// TwinCAT 3 PLC project Heatpump
// ProgramVersion: 3.1.4026.11
// libraries:
//   Tc2_Math, * (Beckhoff Automation GmbH)
//   Tc2_Standard, * (Beckhoff Automation GmbH)
//   Tc2_System, * (Beckhoff Automation GmbH)
//   Tc2_Utilities, * (Beckhoff Automation GmbH)
// project tree:
//   DUTs/ E_Event.TcDUT, E_EventType.TcDUT, E_LogType.TcDUT, E_Severity.TcDUT, E_State.TcDUT, ST_ConfigValues.TcDUT, ST_Event.TcDUT, ST_Events.TcDUT, ST_ErrorEvents.TcDUT, ST_LogBuffer.TcDUT, ST_LogEntry.TcDUT, ST_WarningEvents.TcDUT, ST_SensorRaw.TcDUT, ST_Actor.TcDUT, ST_FailureMessage.TcDUT, ST_Incident.TcDUT, ST_ProcessData.TcDUT, E_FailureLevel.TcDUT, ST_Sensor.TcDUT
//   GVLs/ GVL.TcGVL
//   / PlcTask.TcTTO
//   POUs/ FB_CoolDownState.TcPOU, FB_ErrorState.TcPOU, FB_IdleState.TcPOU, FB_OffState.TcPOU, FB_ProcessData.TcPOU, FB_RunningState.TcPOU, FB_StartWaterFlowState.TcPOU, FB_StateMachine.TcPOU, I_State.TcIO, MAIN.TcPOU
//   POUs/utils/ calculateTargetTemperatureOn.TcPOU, calculateTargetTemperatureOff.TcPOU, convertTimerToDisplayValue.TcPOU, isVentilOpen.TcPOU, LogMessage.TcPOU, setEventInfo.TcPOU, resetApplication.TcPOU, ScaleAndRound.TcPOU, ScaleAndRoundString.TcPOU, switchWaterVentil.TcPOU, toErrorText.TcPOU, toggleIntermediateCircuitPump.TcPOU, togglePvBoost.TcPOU, transitionToErrorState.TcPOU, clearErrorList.TcPOU, updateEventWithTimestamp.TcPOU, UpdateLogTimestampWithSystemTime.TcPOU
// real-time tasks:
//   TASK PlcTask: cycle T#10ms, priority 1, ADS port 350
// I/O:
//   DEVICE Gerät 1 (EtherCAT), AmsNetId 5.124.202.224.2.1
//     Klemme 10 (EK1200) [EK1200-5000 EtherCAT Netzteil (2A E-Bus)]
//       Klemme 2 (EL3152) [EL3152 2K. Ana. Eingang 4-20mA]
//       Klemme 3 (EL2004) [EL2004 4K. Dig. Ausgang 24V, 0.5A]
//       Klemme 4 (EL3204) [EL3204 4K. Ana. Eingang PT100 (RTD)]
//       Klemme 5 (EL3102) [EL3102 2K. Ana. Eingang +/-10V, Diff.]
//       Klemme 6 (EL1008) [EL1008 8K. Dig. Eingang 24V, 3ms]
//       Klemme 18 (EL1008) [EL1008 8K. Dig. Eingang 24V, 3ms]
//       Klemme 7 (EL3204) [EL3204 4K. Ana. Eingang PT100 (RTD)]
//       Klemme 9 (EL2622) [EL2622 2K. Relais Ausgang, Schließer (230V AC / 30V DC)]
//       Klemme 8 (EL2622) [EL2622 2K. Relais Ausgang, Schließer (230V AC / 30V DC)]
//       Klemme 19 (EL3204) [EL3204 4K. Ana. Eingang PT100 (RTD)]
//       Klemme 20 (EL9011) [EL9011 Endklemme]
// variable links:
//   Heatpump/Heatpump Instance <-> Device 1 (EtherCAT)/Term 10 (EK1200)/Term 18 (EL1008)
//     PlcTask Inputs/MAIN.pd.incident.incidentFlowIntermediateCircuit <-> Channel 1/Input
//   Heatpump/Heatpump Instance <-> Device 1 (EtherCAT)/Term 10 (EK1200)/Term 19 (EL3204)
//     PlcTask Inputs/MAIN.fbProcessdata.sensorRaw.temperatureSourceWaterIn <-> RTD Inputs Channel 1/Value
//     PlcTask Inputs/MAIN.fbProcessdata.sensorRaw.temperatureSourceWaterOut <-> RTD Inputs Channel 2/Value
//   Heatpump/Heatpump Instance <-> Device 1 (EtherCAT)/Term 10 (EK1200)/Term 2 (EL3152)
//     PlcTask Inputs/MAIN.fbProcessdata.sensorRaw.pressureHigh <-> Channel 1/Value
//     PlcTask Inputs/MAIN.fbProcessdata.sensorRaw.pressureLow <-> Channel 2/Value
//   Heatpump/Heatpump Instance <-> Device 1 (EtherCAT)/Term 10 (EK1200)/Term 3 (EL2004)
//     PlcTask Outputs/MAIN.pd.actor.operatingStateCompressor <-> Channel 1/Output
//     PlcTask Outputs/MAIN.pd.actor.operatingStateLed <-> Channel 3/Output
//     PlcTask Outputs/MAIN.pd.actor.operatingStateWaterPump <-> Channel 2/Output
//   Heatpump/Heatpump Instance <-> Device 1 (EtherCAT)/Term 10 (EK1200)/Term 4 (EL3204)
//     PlcTask Inputs/MAIN.fbProcessdata.sensorRaw.temperatureEvaporatingIn <-> RTD Inputs Channel 2/Value
//     PlcTask Inputs/MAIN.fbProcessdata.sensorRaw.temperatureEvaporatingOut <-> RTD Inputs Channel 1/Value
//     PlcTask Inputs/MAIN.fbProcessdata.sensorRaw.temperatureFlow <-> RTD Inputs Channel 3/Value
//     PlcTask Inputs/MAIN.fbProcessdata.sensorRaw.temperatureReturn <-> RTD Inputs Channel 4/Value
//   Heatpump/Heatpump Instance <-> Device 1 (EtherCAT)/Term 10 (EK1200)/Term 5 (EL3102)
//     PlcTask Inputs/MAIN.fbProcessdata.sensorRaw.pressureDifferenceEvaporator <-> Channel 1/Value
//   Heatpump/Heatpump Instance <-> Device 1 (EtherCAT)/Term 10 (EK1200)/Term 6 (EL1008)
//     PlcTask Inputs/MAIN.pd.incident.alarmExpansionValve <-> Channel 3/Input
//     PlcTask Inputs/MAIN.pd.incident.incidentCompressor <-> Channel 5/Input
//     PlcTask Inputs/MAIN.pd.incident.incidentHighPressure <-> Channel 7/Input
//     PlcTask Inputs/MAIN.pd.incident.incidentLowPressure <-> Channel 8/Input
//     PlcTask Inputs/MAIN.pd.incident.incidentWaterFlow <-> Channel 6/Input
//     PlcTask Inputs/MAIN.pd.sensor.boilerHeatRequest <-> Channel 2/Input
//     PlcTask Inputs/MAIN.pd.sensor.photovoltaicSurplus <-> Channel 4/Input
//     PlcTask Inputs/MAIN.pd.sensor.userConfirmation <-> Channel 1/Input
//   Heatpump/Heatpump Instance <-> Device 1 (EtherCAT)/Term 10 (EK1200)/Term 7 (EL3204)
//     PlcTask Inputs/MAIN.fbProcessdata.sensorRaw.boilerTemperature <-> RTD Inputs Channel 4/Value
//     PlcTask Inputs/MAIN.fbProcessdata.sensorRaw.bufferMiddleTemperature <-> RTD Inputs Channel 2/Value
//     PlcTask Inputs/MAIN.fbProcessdata.sensorRaw.bufferTopTemperature <-> RTD Inputs Channel 3/Value
//     PlcTask Inputs/MAIN.fbProcessdata.sensorRaw.temperatureOverheatedGas <-> RTD Inputs Channel 1/Value
//   Heatpump/Heatpump Instance <-> Device 1 (EtherCAT)/Term 10 (EK1200)/Term 8 (EL2622)
//     PlcTask Outputs/MAIN.pd.actor.operatingStateIntermediateCircuitPump <-> Channel 1/Output
//   Heatpump/Heatpump Instance <-> Device 1 (EtherCAT)/Term 10 (EK1200)/Term 9 (EL2622)
//     PlcTask Outputs/MAIN.pd.actor.closeFlowVentil <-> Channel 1/Output
//     PlcTask Outputs/MAIN.pd.actor.openFlowVentil <-> Channel 2/Output

CONFIGURATION Heatpump
    RESOURCE PLC ON TwinCAT3
        TASK PlcTask(INTERVAL := T#1ms, PRIORITY := 4);
        PROGRAM MAIN WITH PlcTask : MAIN;
    END_RESOURCE
END_CONFIGURATION

// ---- DUTs/E_Event.TcDUT
{attribute 'qualified_only'}
{attribute 'strict'}
TYPE E_Event :
(
	SwitchOn := 0,
	SwitchOff := 1,
	HeatIsRequested := 2,
	HeatTemperaturreached := 3,
	CooledDown := 4,
	Confirmed := 5
);
END_TYPE

// ---- DUTs/E_EventType.TcDUT
{attribute 'qualified_only'}
{attribute 'strict'}
TYPE E_EventType :
(
	None								:= 0,
	(* Normal StateMachine changes *)	
	SwitchOn 							:= 1,
	SwitchOff 							:= 2,
	HeatIsRequested 					:= 3,
	TargetTemperatureReached 			:= 4,
	CooledDown 							:= 5,
	Confirm 							:= 6,
	minWaterFlowReached					:= 7,
	
	(* Errors *)
	PressureDiffEvaporatorTooHigh		:= 101,
	EvaporatingTemperatureTooLow		:= 102,
	EvaporatingFlowRateTooLow			:= 103,
	LowPressureRefrigerationThermostat	:= 104,
	HighPressureRefrigerationThermostat	:= 105,
	MotorProtectionTriggered			:= 106,
	ExpansionValveTriggered				:= 107,
	IntermediateCircuitFlowRateTooLow	:= 108,
	LowPressureRefrigerationCalc		:= 109,
	TemperatureSourceWaterOutMinTooLow  := 110,
		
	(* Warnings *)
	HighPressureRefrigerationCalc		:= 202,
	WaterTankLevelTooLow				:= 203,
	WaterTankDataMissing				:= 204
);
END_TYPE

// ---- DUTs/E_LogType.TcDUT
{attribute 'qualified_only'}
{attribute 'strict'}
TYPE E_LogType :
(
    INFO := 0,
    WARNING := 1,
    ERROR := 2
);
END_TYPE

// ---- DUTs/E_Severity.TcDUT
{attribute 'qualified_only'}
{attribute 'strict'}
TYPE E_Severity :
(
	Error := 0,
	Warning := 1,
	Event := 2
);
END_TYPE

// ---- DUTs/E_State.TcDUT
{attribute 'qualified_only'}
{attribute 'strict'}
TYPE E_State :
(
	OFF := 0,
	IDLE := 1,
	START_WATER_FLOW := 2,
	RUNNING := 3,
	COOLDOWN := 4,
    ERROR := 5
);
END_TYPE

// ---- DUTs/ST_ConfigValues.TcDUT
TYPE ST_ConfigValues :
STRUCT	
	targetTemperatureOn 			:	REAL	:= 	33; 	// Einschalttemperatur bei deren Unterschreiten die Waermepumpe eingeschaltet wird
	targetTemperatureOnPV 			:	REAL	:= 	40; 	// Bei PV-Überschuss: Einschalttemperatur bei deren Unterschreiten die Waermepumpe eingeschaltet wird
	targetTemperatureOff 			:	REAL	:= 	41; 	// Auschaltemperatur bei deren Ueberschreiten die Waermepume ausgeschaltet wird	
	targetTemperatureOffPV			:	REAL	:= 	50; 	// Bei PV-Überschuss: Auschaltemperatur bei deren Ueberschreiten die Waermepume ausgeschaltet wird	
	maxReturnTemperature			:	REAL	:= 	53; 	// Schaltet aus / nicht ein, falls Rücklauf Temperatur zu hoch, z.B. wenn Holzkessel heizt
	minIdleSec 						:	TIME 	:= 	T#10M;	// Minimale Auschalt-Dauer (verhindert haeufiges Einschalten) [Minuten]
	temperatureDiffBacklashOff 		:	REAL	:= 	1.0; 	// Temperaturdifferenz zwischen Vorlauf und Rücklauf, bei dessen Unterschreiten die Wasserpumpe ausgeschaltet wird
	temperatureDiffBoilerLaden 		:	REAL	:= 	4.0; 	// Temperaturdifferenz zwischen Puffer oben und Boiler, die unterschritten sein muss, damit die Wärmepumpe einschaltet.

	// Limits*)
	pressureHighMax 				:	REAL	:= 	16; 	// Maximaler Druck auf der Hochdruckseite [bar]
	pressureLowMin 					:	REAL	:= 	0.4; 	// Minimaler Druck auf der Niederdruckseite [bar]. Entspricht -5°C. Falls niedriger deutet dies auf ein Kältemittel-Leck hin 
	pressureDifferenceEvaporatorMax :	REAL 	:= 	45;		// Maximaler Druckverlust des Verdampfer-Wärmetauschers [mbar]
	evaporatingTemperatureOutMin 	:	REAL 	:=	1.0; 	// Minimale Temperatur am Austritt des Verdampfer-Wärmetausschers. Triplepunkt des Wassers. [°C]	
	temperatureSourceWaterOutMin	:	REAL 	:=	2.3;  	// Minimale Temperatur am Quellasser-Austritt des Zwischenkreis-Wärmetausschers. Triplepunkt des Wassers. [°C]
END_STRUCT
END_TYPE

// ---- DUTs/ST_Event.TcDUT
TYPE ST_Event :
STRUCT
	eventType		: E_EventType := E_EventType.None;
	severity 		: E_Severity := E_Severity.Event;
	isTriggered		: BOOL := FALSE;
	isSelfHealing   : BOOL := FALSE;  	// selbst heilend: Nach einem Error und automatischem Beheben der Ursache startet die WP wieder
	message	 		: STRING(255);
	timestamp 		: DATE_AND_TIME;
END_STRUCT
END_TYPE

// ---- DUTs/ST_Events.TcDUT
TYPE ST_Events :
STRUCT
	(* Normal StateMachine changes *)
	switchOff 							: ST_Event := (eventType := E_EventType.SwitchOff);  
	switchOn 							: ST_Event := (eventType := E_EventType.SwitchOn);  
	confirmed							: ST_Event := (eventType := E_EventType.Confirm);
	heatIsRequested 					: ST_Event := (eventType := E_EventType.HeatIsRequested);  
	targetTemperatureReached			: ST_Event := (eventType := E_EventType.TargetTemperatureReached);
	cooledDown							: ST_Event := (eventType := E_EventType.CooledDown);
	minWaterFlowReached					: ST_Event := (eventType := E_EventType.MinWaterFlowReached);
		
	(* Errors *)
     errorEvents						: ST_ErrorEvents; 
	 errorsDetected						: BOOL := FALSE;

	(* Warnings *)
	warningEvents						:ST_WarningEvents;
END_STRUCT
END_TYPE

// ---- DUTs/ST_ErrorEvents.TcDUT
TYPE ST_ErrorEvents :
	STRUCT
		(* Errors *)
		PressureDiffEvaporatorTooHigh		: ST_Event := (eventType := E_EventType.PressureDiffEvaporatorTooHigh, isSelfHealing:=FALSE, severity:= E_Severity.Error, message := 'Druckdifferenz am Verdampfer zu hoch. Einfriergefahr');  
		EvaporatingTemperatureTooLow		: ST_Event := (eventType := E_EventType.EvaporatingTemperatureTooLow, isSelfHealing:=TRUE, severity:= E_Severity.Error, message := 'Autrittstemperatur zu niedrig');  
		EvaporatingFlowRateTooLow			: ST_Event := (eventType := E_EventType.EvaporatingFlowRateTooLow, isSelfHealing:=TRUE, severity:= E_Severity.Error, message := 'Durchflussmenge zu niedrig');  
		LowPressureRefrigerationThermostat	: ST_Event := (eventType := E_EventType.LowPressureRefrigerationThermostat, isSelfHealing:=FALSE, severity:= E_Severity.Error, message := 'Thermostat: Niederdruck zu niedrig');  
		HighPressureRefrigerationThermostat	: ST_Event := (eventType := E_EventType.HighPressureRefrigerationThermostat, isSelfHealing:=FALSE, severity:= E_Severity.Error, message := 'Thermostat: Hochdruck zu hoch');  
		MotorProtectionTriggered			: ST_Event := (eventType := E_EventType.MotorProtectionTriggered, isSelfHealing:=FALSE, severity:= E_Severity.Error, message := 'Motorschutzschalter hat ausgelöst');  
		ExpansionValveTriggered				: ST_Event := (eventType := E_EventType.ExpansionValveTriggered, isSelfHealing:=FALSE, severity:= E_Severity.Error, message := 'Expansionsventil ausgelöst');
		IntermediateCircuitFlowRateTooLow	: ST_Event := (eventType := E_EventType.IntermediateCircuitFlowRateTooLow, isSelfHealing:=TRUE, severity:= E_Severity.Error, message := 'Sole Durchflussmenge im Zwischenkreis zu niedrig');
		LowPressureRefrigerationCalc		: ST_Event := (eventType := E_EventType.LowPressureRefrigerationCalc, isSelfHealing:=FALSE, severity:= E_Severity.Error, message := 'Sensor: Niederdruck zu niedrig');  
		TemperatureSourceWaterOutMinTooLow	: ST_Event := (eventType := E_EventType.TemperatureSourceWaterOutMinTooLow, isSelfHealing:=TRUE, severity:= E_Severity.Error, message := 'Quellwasser-Autrittstemperatur zu niedrig. Einfriergefahr');  
	END_STRUCT
END_TYPE

// ---- DUTs/ST_LogBuffer.TcDUT
TYPE ST_LogBuffer :
STRUCT
    aEntries : ARRAY[1..100] OF ST_LogEntry;
END_STRUCT
END_TYPE

// ---- DUTs/ST_LogEntry.TcDUT
TYPE ST_LogEntry :
STRUCT
    sMessage : STRING(255);
    dtTimestamp : DATE_AND_TIME;
    eType : E_LogType;
	sTypeName : STRING(20);
END_STRUCT
END_TYPE

// ---- DUTs/ST_WarningEvents.TcDUT
TYPE ST_WarningEvents :
STRUCT
	(* Warnings *)
	HighPressureRefrigerationCalc		: ST_Event := (eventType := E_EventType.HighPressureRefrigerationCalc, severity:= E_Severity.Warning, message := 'Sensor: Niederdruck zu hoch');  
	WaterTankLevelTooLow				: ST_Event := (eventType := E_EventType.WaterTankLevelTooLow, severity:= E_Severity.Warning, message := 'Wasserstand des Tanks (Quelle) zu niedrig');  
	WaterTankDataMissing				: ST_Event := (eventType := E_EventType.WaterTankDataMissing, severity:= E_Severity.Warning, message := 'Tanksensor (Quelle) sendet keine Daten mehr');  
END_STRUCT
END_TYPE

// ---- DUTs/ST_SensorRaw.TcDUT
TYPE ST_SensorRaw :
    STRUCT
		(* EL3204 - 1*)
        temperatureEvaporatingOut		AT %I*	: INT;  (* Verdampfungstemperatur in °C (Ausgang) *)
        temperatureEvaporatingIn		AT %I*	: INT;  (* Verdampfungstemperatur in °C (Eingang) *)
        temperatureFlow	 				AT %I*	: INT;  (* Vorlauftemperatur in °C *)
        temperatureReturn				AT %I*	: INT;  (* Rücklauftemperatur in °C *)
		
		(* EL3204 - 2*)
        temperatureOverheatedGas		AT %I*	: INT;  (* Saugtemperatur des überhitzten Gases *)
        bufferTopTemperature			AT %I*	: INT;  (* Temperatur des Puffers oben in °C *)
		bufferMiddleTemperature			AT %I*	: INT;  (* Temperatur des Puffers in der Mitte °C *)	
		boilerTemperature				AT %I*	: INT;  (* Boiler-Temperatur oben °C *)	
		
		(* EL3204 - 3*)
		temperatureSourceWaterIn		AT %I*	: INT;  (* Quellwassertemperatur Eingang in °C *)
		temperatureSourceWaterOut		AT %I*	: INT;  (* Quellwassertemperatur Ausgang in °C *)		

		(* EL3122 - 4-20mA*)
        pressureHigh					AT %I*	: INT;  (* Hochdruck Kältekreis in bar *)
        pressureLow						AT %I*	: INT;  (* Niederdruck Kältekreis in bar *)
		
		(* EL3064 - 0-10V* or EL3102 -  +/-10V *)
        pressureDifferenceEvaporator	AT %I*	: INT;  (* Druckdifferenz im Verdampfer in mbar *)
    END_STRUCT
END_TYPE

// ---- DUTs/ST_Actor.TcDUT
TYPE ST_Actor :
    STRUCT
		(* EL2004 - Digital Out*)
        operatingStateCompressor 				AT %Q* : BOOL := FALSE;  // Status des Verdichters: Ein/Aus
        operatingStateWaterPump 				AT %Q* : BOOL := FALSE;  // Status der Heizungspumpe: Ein/Aus
        operatingStateIntermediateCircuitPump 	AT %Q* : BOOL := FALSE;  // Status der Heizungspumpe: Ein/Aus
		operatingStateLed						AT %Q* : BOOL := FALSE;  // LED am Schaltschrank, die anzeigt ob die Wärmepumpe eingschaltet/bereit ist
		openFlowVentil   						AT %Q* : BOOL := FALSE;  // Wasserventil öffnen
		closeFlowVentil   						AT %Q* : BOOL := FALSE;  // Wasserventil schliessen 
    END_STRUCT
END_TYPE

// ---- DUTs/ST_FailureMessage.TcDUT
TYPE ST_FailureMessage :
    STRUCT
        message: STRING[100];  (* Fehlermeldung *)
        level: E_FailureLevel;  (* Fehlerstufe *)
    END_STRUCT
END_TYPE

// ---- DUTs/ST_Incident.TcDUT
TYPE ST_Incident :
    STRUCT
		// Connected to IO Klemmen		
        alarmExpansionValve				AT %I*			: BOOL;		// Alarm: Elektronisches Expansionsventil - EL1008.3
        incidentCompressor				AT %I*			: BOOL; 	// Störung: Verdichter / Motorschutzschalter - EL1008.5
        incidentWaterFlow				AT %I*			: BOOL; 	// Störung: Quellwasser-Durchfluss zu niedrig - EL1008.6  Achtung!!! invertiert: True bedeutet genug Fluss vorhanden
        incidentFlowIntermediateCircuit	AT %I*			: BOOL; 	// Störung: Durchfluss im Verdampfer (Zwischenkreis) zu niedrig. Achtung!!! invertiert: True bedeutet genug Fluss vorhanden 
        incidentHighPressure			AT %I*			: BOOL; 	// Störung: Hochdruck zu hoch - EL1008.7
        incidentLowPressure				AT %I*			: BOOL; 	// Störung: Niederdruck zu niedrig - EL1008.8 

		// Calculated from Business Logic
        incidentTankLevelTooLow					: BOOL;  // Störung: Wasserstand des Tanks zu niedrig 
        incidentTankSensorDataMissing			: BOOL;  // Störung: Tanksensor sendet keine Daten mehr 
    END_STRUCT
END_TYPE

// ---- DUTs/ST_ProcessData.TcDUT
TYPE ST_ProcessData :
    STRUCT
        id					: STRING[50];  (* Äquivalent zu String in Java *)
        timestamp			: TIME;  (* Äquivalent zu Instant in Java *)
        sensor				: ST_Sensor;  (* Instanz von Sensor *)
        actor				: ST_Actor;  (* Instanz von Actor *)
        incident			: ST_Incident;  (* Instanz von Incident *)
        waitCounter			: INT;  (* Integer *)
        messages			: ARRAY[1..10] OF ST_FailureMessage;  (* Set als Array, maximale Anzahl definieren *)
    END_STRUCT
END_TYPE

// ---- DUTs/E_FailureLevel.TcDUT
{attribute 'qualified_only'}
{attribute 'strict'}
{attribute 'to_string'}
TYPE E_FailureLevel :
( 
    ERROR := 0,
    WARNING := 1,
    INFO := 2
);
END_TYPE

// ---- DUTs/ST_Sensor.TcDUT
TYPE ST_Sensor :
    STRUCT
        temperatureEvaporatingIn				: REAL;  // Verdampfungstemperatur in °C (Eingang)
        temperatureEvaporatingOut				: REAL;  // Verdampfungstemperatur in °C (Ausgang)
        temperatureFlow	 						: REAL;  // Vorlauftemperatur in °C
        temperatureReturn						: REAL;  // Rücklauftemperatur in °C
        bufferTopTemperature					: REAL;  // Temperatur des Puffers oben in °C
        bufferMiddleTemperature					: REAL;  // Temperatur des Puffers in der Mitte °C		
		boilerTemperature						: REAL;  // Boiler-Temperatur oben °C
        temperatureOverheatedGas				: REAL;  // Saugtemperatur des überhitzten Gases
        temperatureSourceWaterIn				: REAL;  // Quellwassertemperatur Eingang in °C
        temperatureSourceWaterOut				: REAL;  // Quellwassertemperatur Ausgang in °C
        pressureHigh							: REAL;  // Hochdruck Kältekreis in bar
        pressureLow								: REAL;  // Niederdruck Kältekreis in bar
        pressureDifferenceEvaporator			: REAL;  // Druckdifferenz im Verdampfer in mbar
        calculatedOverheatTemperature			: REAL;  // Berechnete Überhitzungstemperatur
        boilerHeatRequest				AT %I*	: BOOL;  // Boiler LadePumpe ist eingeschaltet - EL1008.1*)
        userConfirmation				AT %I*	: BOOL;  // Taster für Ein-/Aus-Quittierung - EL1008.2*) 
		photovoltaicSurplus				AT %I*	: BOOL;  // Photovoltaik Überschuss - gemeldet vom PV-WechselrichterEL1008.4*)
		photovoltaicBoost				  		: BOOL;  // Photovoltaik Boost - ist kein Sensor - sondern per Click einschaltbar*)
    END_STRUCT
END_TYPE

// ---- GVLs/GVL.TcGVL
{attribute 'qualified_only'}
VAR_GLOBAL PERSISTENT
	configValues			:   ST_ConfigValues;			// Konfigurationsparaeter - Müssen vom User geändert werden können
END_VAR
VAR_GLOBAL 
	lastErrorsOccurred		:   ARRAY[0..6] OF ST_Event;  	// List of last errors occurred
	g_LogData : ST_LogBuffer;
END_VAR

// ---- POUs/I_State.TcIO
INTERFACE I_State

PROPERTY Description : STRING
GET
END_GET
END_PROPERTY

METHOD ErrorDetected : BOOL
VAR_IN_OUT
	errorEvents		: ST_ErrorEvents;
END_VAR
END_METHOD

METHOD HeatIsRequested : BOOL
VAR_INPUT
END_VAR
END_METHOD

METHOD MinWaterFlowReached : BOOL
VAR_INPUT
END_VAR
END_METHOD

PROPERTY Name : String
GET
END_GET
END_PROPERTY

PROPERTY State : E_State
GET
END_GET
END_PROPERTY

METHOD TargetTemperatureReached : BOOL
VAR_INPUT
END_VAR
END_METHOD

METHOD UserPressedConfirmationButton : BOOL
VAR_INPUT
END_VAR
END_METHOD

METHOD UserPressedSwitchOffButton : BOOL
VAR_INPUT
END_VAR
END_METHOD

METHOD UserPressedSwitchOnButton : BOOL
VAR_INPUT
END_VAR
END_METHOD

METHOD WaterHasCooledDown : BOOL
VAR_INPUT
END_VAR
END_METHOD

END_INTERFACE

// ---- POUs/MAIN.TcPOU
PROGRAM MAIN
VAR
	fbStateMachine				:	FB_StateMachine;
	fbProcessdata				:   FB_Processdata;
	pd 							: 	ST_ProcessData;	
END_VAR

fbProcessdata(pd := pd);

fbStateMachine(pd := pd);

END_PROGRAM

// ---- POUs/FB_StateMachine.TcPOU
FUNCTION_BLOCK FB_StateMachine
VAR_INPUT	
	pd 							: 	REFERENCE TO ST_ProcessData;
END_VAR
VAR_OUTPUT
	iState						:	I_State := fbOffState;	
	events						:	ST_Events();
	defaultEvents 				: 	ST_Events();  			// leere Kopie
END_VAR
VAR
	fbOffState					:	FB_OffState(THIS);
	fbIdleState					:	FB_IdleState(THIS);
	fbStartWaterFlowState		:	FB_StartWaterFlowState(THIS);
	fbRunningState				:	FB_RunningState(THIS);
	fbCoolDownState				:	FB_CoolDownState(THIS);
	fbErrorState				:	FB_ErrorState(THIS);
	timerTON 					: 	TON;             		// TON-Timer
	
	bStartButtonPressed    				: 	BOOL;
	bStopButtonPressed					: 	BOOL;	
    bClearErrorListButton				:   BOOL;  		
    bToggleButtonVentil 				: 	BOOL; 	
	bToggleIntermediateCircuitPump		: 	BOOL; 	
	bToggleButtonPvBoost				: 	BOOL; 
	rtrigButtonSwitchOn					:	R_TRIG;
	rtrigButtonSwitchOff				:	R_TRIG;
	rtrigButtonConfirmation				:	R_TRIG;	
	rtrigClearErrorListButton			:	R_TRIG;
	rtrigToggleButtonVentil				:   R_TRIG;		// rising Edge
	rtrigToggleIntermediateCircuitPump	:   R_TRIG;		
	rtrigToogleButtonPvBoost			:   R_TRIG;	
	strState							: 	STRING;
	strInfotext							: 	STRING(256);
	
	isStartButtonEnabled		:	BOOL 	:=	TRUE;
	isStopButtonEnabled			:	BOOL 	:=	TRUE;
	timerValueToDisplay			:	INT		:= 	0;	
	bIsTimerVisible				: 	BOOL	:=  FALSE;
END_VAR

rtrigButtonSwitchOn(CLK := bStartButtonPressed);
rtrigButtonSwitchOff(CLK := bStopButtonPressed);
rtrigButtonConfirmation(CLK := pd.sensor.userConfirmation);
rtrigClearErrorListButton(CLK := bClearErrorListButton);
rtrigToggleButtonVentil(CLK := bToggleButtonVentil);
rtrigToggleIntermediateCircuitPump(CLK := bToggleIntermediateCircuitPump);
rtrigToogleButtonPvBoost(CLK := bToggleButtonPvBoost);

timerTON();

// Zuweisung von defaultEvent zu myEvent (Wertkopie)
events := defaultEvents;

generateEvents(events);

IF events.errorsDetected THEN
	iState.ErrorDetected(events.errorEvents);
ELSE IF iState.State = E_State.ERROR THEN
		LogMessage(E_LogType.WARNING, 'Fehler steht nicht mehr an ->', idleState.Name);
		SetState(idleState);
	END_IF	
END_IF 

IF events.switchOff.isTriggered THEN
	iState.UserPressedSwitchOffButton();
END_IF 

IF events.switchOn.isTriggered THEN
	iState.UserPressedSwitchOnButton();
END_IF 

IF events.confirmed.isTriggered THEN
	iState.UserPressedConfirmationButton();
END_IF 

IF events.heatIsRequested.isTriggered THEN
	iState.HeatIsRequested();
END_IF 

IF events.targetTemperatureReached.isTriggered THEN
	iState.TargetTemperatureReached();
END_IF 

IF events.cooledDown.isTriggered THEN
	iState.WaterHasCooledDown();
END_IF

IF events.minWaterFlowReached.isTriggered THEN
	iState.MinWaterFlowReached();
END_IF

IF rtrigClearErrorListButton.Q THEN
	clearErrorList();
END_IF

IF rtrigToggleButtonVentil.Q THEN
	switchWaterVentil(NOT isVentilOpen(pd), THIS);
END_IF

IF rtrigToggleIntermediateCircuitPump.Q THEN
	toggleIntermediateCircuitPump(THIS);
END_IF

IF rtrigToogleButtonPvBoost.Q THEN
	togglePvBoost(THIS);
END_IF


setLabelText();
setButtonState();

timerTON();
timerValueToDisplay := convertTimerToDisplayValue(timerTON);

IF iState.State = E_State.IDLE AND timerTON.IN = TRUE AND timerTON.Q = FALSE THEN 	
	bIsTimerVisible := TRUE;
ELSE
	bIsTimerVisible := FALSE;
END_IF

PROPERTY INTERNAL CoolDownState : I_State
GET
CoolDownState := THIS^.fbCoolDownState;
END_GET
END_PROPERTY

PROPERTY INTERNAL ErrorState : I_State
GET
ErrorState := THIS^.fbErrorState;
END_GET
END_PROPERTY

//FB_Init ist immer implizit verfügbar und wird primär für die Initialisierung verwendet.
//Der Rückgabewert wird nicht ausgewertet. Für gezielte Einflussnahme können Sie
//die Methoden explizit deklarieren und darin mit dem Standard-Initialisierungscode 
//zusätzlichen Code bereitstellen. Sie können den Rückgabewert auswerten.
METHOD FB_Init: BOOL
VAR_INPUT    
	bInitRetains: BOOL; // TRUE: Die Retain-Variablen werden initialisiert (Reset warm / Reset kalt)    
	bInCopyCode: BOOL;  // TRUE: Die Instanz wird danach in den Kopiercode kopiert (Online-Change)
END_VAR
END_METHOD

METHOD generateEvents : BOOL
VAR_IN_OUT
	events					:	ST_Events();
END_VAR
IF (rtrigButtonSwitchOff.Q OR (rtrigButtonConfirmation.Q AND (iState.State <> E_State.OFF OR iState.State = E_State.ERROR))) THEN
	events.switchOff.isTriggered := TRUE;
ELSIF (rtrigButtonSwitchOn.Q OR (rtrigButtonConfirmation.Q AND iState.State = E_State.OFF)) THEN
	events.switchOn.isTriggered := TRUE;
ELSIF (isHeatRequested()) THEN
	events.heatIsRequested.isTriggered := TRUE;
ELSIF ((pd.sensor.temperatureFlow - pd.sensor.temperatureReturn) < GVL.configValues.temperatureDiffBacklashOff
	AND (pd.sensor.temperatureEvaporatingIn - pd.sensor.temperatureEvaporatingOut) < GVL.configValues.temperatureDiffBacklashOff 
	AND iState.State = E_State.COOLDOWN) THEN
		events.cooledDown.isTriggered := TRUE;
ELSIF (isTargetTemperatureReached()) THEN
	events.targetTemperatureReached.isTriggered := TRUE;
ELSIF (pd.incident.incidentWaterFlow AND      				// Durchfluss Quellwasser ist ok
	pd.incident.incidentFlowIntermediateCircuit AND			// Durchfluss Sole im Zwischenkreis ist ok
	iState.State = E_State.START_WATER_FLOW) THEN
	events.minWaterFlowReached.isTriggered := TRUE;
END_IF

//***** Errors *****

(* Prüfe minimalen Druck auf der Niederdruckseite über Ranco Thermostat [bar] *)
IF pd.incident.incidentLowPressure THEN
	setEventInfo(events, events.errorEvents.LowPressureRefrigerationThermostat, TRUE, CONCAT('Ranco Thermostat: zu niedriger Niederdruck [bar]: ', ScaleAndRoundString(pd.sensor.pressureLow, 10))); 
END_IF

(*Prüfe maximalen Druck auf der Hochdruckseite über Ranco Thermostat [bar]  *)
IF pd.incident.incidentHighPressure THEN
	setEventInfo(events, events.errorEvents.HighPressureRefrigerationThermostat, TRUE, CONCAT('Ranco Thermostat: zu hoher Hochdruck [bar]: ', ScaleAndRoundString(pd.sensor.pressureHigh, 10)));
END_IF

(* Motor-Schutzschalter hat ausgelöst *)
IF pd.incident.incidentCompressor THEN
	setEventInfo(events, events.errorEvents.MotorProtectionTriggered, TRUE, 'Motorschutzschalter hat ausgelöst');
END_IF

(* Expansionsventil meldet Fehler *)
IF pd.incident.alarmExpansionValve THEN
	setEventInfo(events, events.errorEvents.ExpansionValveTriggered, TRUE, 'Expansionsventil meldet Fehler');
END_IF

(* Prüfe Mindest-Druck auf der Niederdruckseite über Druck-Transmitter [bar] *)
IF pd.sensor.PressureLow < GVL.configValues.pressureLowMin THEN
	setEventInfo(events, events.errorEvents.LowPressureRefrigerationCalc, TRUE, CONCAT('Gemessener Niederdruck zu niedrig: [bar]: ', ScaleAndRoundString(pd.sensor.PressureLow, 10)));
END_IF

(* Maximaler Druckverlust des Verdampfer-Wärmetauschers [mbar] *)
IF pd.sensor.PressureDifferenceEvaporator > GVL.configValues.PressureDifferenceEvaporatorMax THEN
	setEventInfo(events, events.errorEvents.PressureDiffEvaporatorTooHigh, TRUE, CONCAT('Druckdifferenz am Verdampfer zu niedrig [mbar]: ', REAL_TO_STRING(REAL_TO_INT(pd.sensor.PressureDifferenceEvaporator))));
END_IF

(* Prüfe minimale Temperatur am Austritt des Verdampfer-Wärmetausschers. *)
IF pd.sensor.TemperatureEvaporatingOut < GVL.configValues.evaporatingTemperatureOutMin THEN
	setEventInfo(events, events.errorEvents.EvaporatingTemperatureTooLow, TRUE, CONCAT('Austritttemperatur am Verdampfer ist zu niedrig [°C]: ', ScaleAndRoundString(pd.sensor.TemperatureEvaporatingOut, 10)));
END_IF

(* Prüfe minimale Temperatur am Quellasser-Austritt des Zwischenkreis-Wärmetausschers. Triplepunkt des Wassers. [°C] *)
IF pd.sensor.temperatureSourceWaterOut < GVL.configValues.temperatureSourceWaterOutMin THEN
	setEventInfo(events, events.errorEvents.TemperatureSourceWaterOutMinTooLow, TRUE, CONCAT('Quellwasser-Autrittstemperatur zu niedrig. Einfriergefahr! [°C]: ', ScaleAndRoundString(pd.sensor.temperatureSourceWaterOut, 10)));
END_IF

(* Prüfe, of Wasser Durchflussmenge ausreichend ist. Mindestens 1800 Liter/Stunde *)
IF NOT pd.incident.incidentWaterFlow AND iState.State = E_State.RUNNING THEN
	setEventInfo(events, events.errorEvents.EvaporatingFlowRateTooLow, TRUE, 'Quellwasser Durchflussmenge zu niedrig');
END_IF

(* Prüfe, of Sole Durchflussmenge im Zwischenkres ausreichend ist. Mindestens 2000 Liter/Stunde *)
IF NOT pd.incident.incidentFlowIntermediateCircuit AND iState.State = E_State.RUNNING THEN
	setEventInfo(events, events.errorEvents.IntermediateCircuitFlowRateTooLow, TRUE, 'Sole Durchflussmenge im Zwischenkreis zu niedrig');
END_IF

// ***** Warnings *****
(* Prüfe maximalen Druck auf der Hochdruckseite [bar] *)
IF pd.sensor.PressureHigh > GVL.configValues.PressureHighMax THEN
	setEventInfo(events, events.warningEvents.HighPressureRefrigerationCalc, FALSE, CONCAT('', ScaleAndRoundString(pd.sensor.PressureHigh, 10)));
ELSE
	events.warningEvents.HighPressureRefrigerationCalc.isTriggered := FALSE;
END_IF

(* TANK_LEVEL_TOO_LOW *)
IF FALSE THEN
	setEventInfo(events, events.warningEvents.WaterTankLevelTooLow, FALSE, 'Wasserstand der Quelle ist zu niedrig');
END_IF

(* TANK_LEVEL Data missing *)
IF FALSE THEN
	setEventInfo(events, events.warningEvents.WaterTankDataMissing, FALSE, 'Keine Daten über den Wasserstand der Quelle verfügbar');
END_IF
END_METHOD

PROPERTY INTERNAL IdleState : I_State
GET
IdleState := THIS^.fbIdleState;
END_GET
END_PROPERTY

METHOD isHeatRequested : BOOL
VAR_INPUT
END_VAR
isHeatRequested := 
	((pd.sensor.bufferTopTemperature < calculateTargetTemperatureOn(pd.sensor.photovoltaicSurplus, pd.sensor.photovoltaicBoost)) OR
	(pd.sensor.boilerHeatRequest = TRUE AND (pd.sensor.bufferTopTemperature <= pd.sensor.boilerTemperature + GVL.configValues.temperatureDiffBoilerLaden)))
	AND iState.State = E_State.IDLE
	AND pd.sensor.temperatureReturn <= GVL.configValues.maxReturnTemperature;
END_METHOD

METHOD isTargetTemperatureReached : BOOL
VAR_INPUT
END_VAR
// In case of State=Running the Heatpump is turned of if following condition are true
isTargetTemperatureReached := 
	((pd.sensor.bufferMiddleTemperature >= calculateTargetTemperatureOff(pd.sensor.photovoltaicSurplus, pd.sensor.photovoltaicBoost)) AND (pd.sensor.boilerHeatRequest = FALSE)	
	  OR pd.sensor.temperatureReturn > GVL.configValues.maxReturnTemperature)
	AND (iState.State = E_State.RUNNING);
END_METHOD

PROPERTY INTERNAL OffState : I_State
GET
OffState := THIS^.fbOffState;
END_GET
END_PROPERTY

PROPERTY INTERNAL RunningState : I_State
GET
RunningState := THIS^.fbRunningState;
END_GET
END_PROPERTY

METHOD setButtonState : BOOL
VAR_INPUT
END_VAR
IF iState.State <> E_State.OFF THEN 
	isStopButtonEnabled := TRUE;
	isStartButtonEnabled := FALSE;
ELSE 
	isStopButtonEnabled := FALSE;
	isStartButtonEnabled := TRUE;
END_IF

bStartButtonPressed				:= FALSE;
bStopButtonPressed				:= FALSE;
bClearErrorListButton 			:= FALSE;
bToggleButtonVentil 			:= FALSE;
bToggleIntermediateCircuitPump	:= FALSE;
bToggleButtonPvBoost			:= FALSE;
END_METHOD

METHOD setLabelText : BOOL
VAR_INPUT
END_VAR
strState := iState.Name;

CASE  iState.State OF 
	E_State.RUNNING:
		strInfotext := CONCAT('Ausschalt-Bedingung:\nDie Ladepumpe ist nicht eingeschaltet   und\ndie Puffertemperatur Mitte ist grösser als ',  ScaleAndRoundString(calculateTargetTemperatureOff(pd.sensor.photovoltaicSurplus, pd.sensor.photovoltaicBoost), 10));
		strInfotext := CONCAT(strInfotext, ' °C');	
	E_State.IDLE:
		strInfotext := CONCAT('Einschalt-Bedingung:\nDie Temperatur am Puffer oben ist niedriger als ',  ScaleAndRoundString(calculateTargetTemperatureOn(pd.sensor.photovoltaicSurplus, pd.sensor.photovoltaicBoost), 10));
		strInfotext := CONCAT(strInfotext, ' °C    oder\ndie Ladepumpe ist ein und der Puffer ist nicht deutlich wärmer als der Boiler');
	E_State.COOLDOWN:
		strInfotext := 'Die Pumpe schaltet aus wenn die Restwärme \naus dem Verflüssiger abtransortiert wurde';
ELSE
	strInfotext := '';	
END_CASE
END_METHOD

METHOD INTERNAL SetState : BOOL
VAR_INPUT
	newState : I_State;
END_VAR
THIS^.iState := newState;
END_METHOD

PROPERTY INTERNAL StartWaterFlowState : I_State
GET
StartWaterFlowState := THIS^.fbStartWaterFlowState;
END_GET
END_PROPERTY

END_FUNCTION_BLOCK

// ---- POUs/FB_OffState.TcPOU
FUNCTION_BLOCK FB_OffState IMPLEMENTS I_State
VAR_INPUT
END_VAR
VAR_OUTPUT
END_VAR
VAR
	pMachine : POINTER TO FB_StateMachine;
END_VAR

PROPERTY Description : STRING
GET
Description := 'Heat pump is switched off';
END_GET
END_PROPERTY

METHOD ErrorDetected : BOOL
VAR_IN_OUT
	errorEvents		: ST_ErrorEvents;
END_VAR

VAR
	message				: STRING(255);
END_VAR
transitionToErrorState(errorEvents := errorEvents, pMachine := pMachine);
END_METHOD

//FB_Init ist immer implizit verfügbar und wird primär für die Initialisierung verwendet.
//Der Rückgabewert wird nicht ausgewertet. Für gezielte Einflussnahme können Sie
//die Methoden explizit deklarieren und darin mit dem Standard-Initialisierungscode 
//zusätzlichen Code bereitstellen. Sie können den Rückgabewert auswerten.
METHOD FB_Init: BOOL
VAR_INPUT    
	bInitRetains: BOOL; // TRUE: Die Retain-Variablen werden initialisiert (Reset warm / Reset kalt)    
	bInCopyCode: BOOL;  // TRUE: Die Instanz wird danach in den Kopiercode kopiert (Online-Change)
	pMachine : POINTER TO FB_StateMachine;
END_VAR
THIS^.pMachine := pMachine;
END_METHOD

METHOD HeatIsRequested : BOOL
END_METHOD

METHOD LimitValuesAreExceeded : BOOL
END_METHOD

METHOD MinWaterFlowReached : BOOL
VAR_INPUT
END_VAR
END_METHOD

PROPERTY Name : STRING
GET
Name := 'aus';
END_GET
END_PROPERTY

PROPERTY State : E_State
GET
State := E_State.OFF;
END_GET
END_PROPERTY

METHOD TargetTemperatureReached : BOOL
END_METHOD

METHOD UserPressedConfirmationButton : BOOL
END_METHOD

METHOD UserPressedSwitchOffButton : BOOL
END_METHOD

METHOD UserPressedSwitchOnButton : BOOL
LogMessage(E_LogType.INFO, 'Einschalt Button wurde gedrückt -> ', pMachine^.IdleState.Name);
pMachine^.pd.actor.operatingStateLed := TRUE;
pMachine^.SetState(pMachine^.IdleState);
END_METHOD

METHOD WaterHasCooledDown : BOOL
END_METHOD

END_FUNCTION_BLOCK

// ---- POUs/utils/transitionToErrorState.TcPOU
FUNCTION transitionToErrorState : BOOL
VAR_IN_OUT
	errorEvents	: ST_ErrorEvents;
END_VAR
VAR_INPUT
	pMachine 	: POINTER TO FB_StateMachine;
END_VAR
VAR
	message		: STRING(255);
	i 			: INT := 0;
END_VAR

pMachine^.pd.actor.operatingStateCompressor := FALSE;
pMachine^.pd.actor.operatingStateWaterPump := FALSE;
pMachine^.pd.actor.operatingStateIntermediateCircuitPump := FALSE;
switchWaterVentil(bOpen := FALSE, pMachine);

IF errorEvents.PressureDiffEvaporatorTooHigh.isTriggered THEN
	GVL.lastErrorsOccurred[i] := errorEvents.PressureDiffEvaporatorTooHigh;
	i := i + 1;
END_IF

IF errorEvents.EvaporatingTemperatureTooLow.isTriggered THEN
	GVL.lastErrorsOccurred[i] := errorEvents.EvaporatingTemperatureTooLow;
	i := i + 1;
END_IF

IF errorEvents.EvaporatingFlowRateTooLow.isTriggered THEN
	GVL.lastErrorsOccurred[i] := errorEvents.EvaporatingFlowRateTooLow;
	i := i + 1;
END_IF

IF errorEvents.IntermediateCircuitFlowRateTooLow.isTriggered THEN
	GVL.lastErrorsOccurred[i] := errorEvents.IntermediateCircuitFlowRateTooLow;
	i := i + 1;
END_IF

IF errorEvents.LowPressureRefrigerationThermostat.isTriggered THEN
	GVL.lastErrorsOccurred[i] := errorEvents.LowPressureRefrigerationThermostat;
	i := i + 1;
END_IF

IF errorEvents.HighPressureRefrigerationThermostat.isTriggered THEN
	GVL.lastErrorsOccurred[i] := errorEvents.HighPressureRefrigerationThermostat;
	i := i + 1;
END_IF


IF errorEvents.LowPressureRefrigerationCalc.isTriggered THEN
	GVL.lastErrorsOccurred[i] := errorEvents.LowPressureRefrigerationCalc;
	i := i + 1;
END_IF

IF errorEvents.MotorProtectionTriggered.isTriggered THEN
	GVL.lastErrorsOccurred[i] := errorEvents.MotorProtectionTriggered;
	i := i + 1;
END_IF

IF errorEvents.ExpansionValveTriggered.isTriggered THEN
	GVL.lastErrorsOccurred[i] := errorEvents.ExpansionValveTriggered;
	i := i + 1;
END_IF

WHILE i <= 6 DO
    GVL.lastErrorsOccurred[i].eventType := E_EventType.None;        // Beispiel für einen "leeren" Event-Typ
    GVL.lastErrorsOccurred[i].severity := E_Severity.Event;         // Standardwert für severity
    GVL.lastErrorsOccurred[i].isTriggered := FALSE;                 // Setzt isTriggered auf FALSE
    GVL.lastErrorsOccurred[i].message := '';                        // Leere Zeichenkette für message
    GVL.lastErrorsOccurred[i].timestamp := DT#1970-01-01-00:00:00;  // Standardzeitstempel (z. B. Unix-Epoche)
    i := i + 1;  
END_WHILE;

message := toErrorText();
LogMessage(E_LogType.ERROR, 'Error detected: ', message);
pMachine^.SetState(pMachine^.ErrorState);

END_FUNCTION

// ---- POUs/utils/switchWaterVentil.TcPOU
FUNCTION switchWaterVentil : BOOL
VAR_INPUT
	bOpen : BOOL; // TRUE = öffnen, FALSE = schließen
	pMachine : POINTER TO FB_StateMachine;
END_VAR

IF (bOpen) THEN
	LogMessage(E_LogType.INFO, 'Betätige Ventil: -> ', 'öffnen');
ELSE
	LogMessage(E_LogType.INFO, 'Betätige Ventil: -> ', 'schliessen');
END_IF;	

IF bOpen THEN
	pMachine^.pd.actor.openFlowVentil := TRUE;
	pMachine^.pd.actor.closeFlowVentil := FALSE;
ELSE
	pMachine^.pd.actor.openFlowVentil := FALSE;
	pMachine^.pd.actor.closeFlowVentil := TRUE;
END_IF

END_FUNCTION

// ---- POUs/utils/LogMessage.TcPOU
FUNCTION LogMessage : BOOL
VAR_INPUT
    eType 		: E_LogType;
	sParam1 	: STRING;
	sParam2  	: STRING;
END_VAR
VAR
    nIndex : INT;
	i : INT;
	sMsg : STRING;
	sTypeName : STRING(20);
END_VAR

sMsg := CONCAT(sParam1, sParam2);

CASE eType OF
    E_LogType.INFO:
        AdsLogStr(ADSLOG_MSGTYPE_HINT, '[INFO] %s', sMsg);
    E_LogType.WARNING:
        AdsLogStr(ADSLOG_MSGTYPE_WARN, '[WARN] %s', sMsg);
    E_LogType.ERROR:
        AdsLogStr(ADSLOG_MSGTYPE_ERROR, '[ERROR] %s', sMsg);
END_CASE

// Schiebe alle bisherigen Einträge um 1 nach unten
FOR i := 100 TO 2 BY -1 DO
	GVL.g_LogData.aEntries[i] := GVL.g_LogData.aEntries[i - 1];
END_FOR;


CASE eType OF
    E_LogType.INFO:    sTypeName := 'INFO';
    E_LogType.WARNING: sTypeName := 'WARNING';
    E_LogType.ERROR:   sTypeName := 'ERROR';
END_CASE;

	
// Eintrag schreiben
// Neuesten Eintrag an Position 1 einfügen
GVL.g_LogData.aEntries[1].sMessage := sMsg;
UpdateLogTimestampWithSystemTime(GVL.g_LogData.aEntries[1]);
GVL.g_LogData.aEntries[1].eType := eType;
GVL.g_LogData.aEntries[1].sTypeName := sTypeName;

LogMessage := TRUE;

END_FUNCTION

// ---- POUs/utils/UpdateLogTimestampWithSystemTime.TcPOU
FUNCTION UpdateLogTimestampWithSystemTime
VAR_INPUT
	stEvent : REFERENCE TO  ST_LogEntry;
END_VAR
VAR
	fbGETSYSTEMTYPE : GETSYSTEMTIME;
	stFileTime : T_FILETIME;
END_VAR

fbGETSYSTEMTYPE(timeLoDW => stFileTime.dwLowDateTime, 
				timeHiDW =>  stFileTime.dwHighDateTime);
				
stEvent.dtTimestamp := FILETIME_TO_DT(fileTime := stFileTime);

END_FUNCTION

// ---- POUs/utils/toErrorText.TcPOU
FUNCTION toErrorText : STRING(255)
VAR
	i				: INT; 
	message			: STRING(255);
	errorArray 		: ARRAY [0..6] OF ST_Event;
END_VAR

FOR i := 0 TO 6 DO
	IF GVL.lastErrorsOccurred[i].isTriggered THEN
		message := CONCAT(message, GVL.lastErrorsOccurred[i].message);
		message := CONCAT(message, ',');
	END_IF
END_FOR

toErrorText := message;

END_FUNCTION

// ---- POUs/FB_IdleState.TcPOU
FUNCTION_BLOCK FB_IdleState IMPLEMENTS I_State
VAR_INPUT
END_VAR
VAR_OUTPUT
END_VAR
VAR
	pMachine : POINTER TO FB_StateMachine;
END_VAR

PROPERTY Description : STRING
GET
Description := 'Heat pump is idle';
END_GET
END_PROPERTY

METHOD ErrorDetected : BOOL
VAR_IN_OUT
	errorEvents		: ST_ErrorEvents;
END_VAR
VAR
	message				: STRING(255);
END_VAR
transitionToErrorState(errorEvents := errorEvents, pMachine := pMachine);
END_METHOD

//FB_Init ist immer implizit verfügbar und wird primär für die Initialisierung verwendet.
//Der Rückgabewert wird nicht ausgewertet. Für gezielte Einflussnahme können Sie
//die Methoden explizit deklarieren und darin mit dem Standard-Initialisierungscode 
//zusätzlichen Code bereitstellen. Sie können den Rückgabewert auswerten.
METHOD FB_Init: BOOL
VAR_INPUT    
	bInitRetains: BOOL; // TRUE: Die Retain-Variablen werden initialisiert (Reset warm / Reset kalt)    
	bInCopyCode: BOOL;  // TRUE: Die Instanz wird danach in den Kopiercode kopiert (Online-Change)
	pMachine : POINTER TO FB_StateMachine;
END_VAR
THIS^.pMachine := pMachine;
END_METHOD

METHOD HeatIsRequested : BOOL
IF pMachine^.timerTON.Q OR NOT pMachine^.timerTON.IN THEN
	LogMessage(E_LogType.INFO, 'Heizung wurde angefordert -> ', pMachine^.StartWaterFlowState.Name);
	pMachine^.timerTON(IN := FALSE);  
    switchWaterVentil(bOpen := TRUE, pMachine);
	pMachine^.pd.actor.operatingStateIntermediateCircuitPump := TRUE;
	pMachine^.SetState(pMachine^.StartWaterFlowState);	
END_IF
END_METHOD

METHOD LimitValuesAreExceeded : BOOL
END_METHOD

METHOD MinWaterFlowReached : BOOL
VAR_INPUT
END_VAR
END_METHOD

PROPERTY Name : STRING
GET
Name := 'bereit';
END_GET
END_PROPERTY

PROPERTY State : E_State
GET
State := E_State.IDLE;
END_GET
END_PROPERTY

METHOD TargetTemperatureReached : BOOL
END_METHOD

METHOD UserPressedConfirmationButton : BOOL
END_METHOD

METHOD UserPressedSwitchOffButton : BOOL
resetApplication(pMachine);
LogMessage(E_LogType.INFO, 'Aus Button wurde gedrückt -> ', pMachine^.OffState.Name);
pMachine^.SetState(pMachine^.OffState);
END_METHOD

METHOD UserPressedSwitchOnButton : BOOL
END_METHOD

METHOD WaterHasCooledDown : BOOL
END_METHOD

END_FUNCTION_BLOCK

// ---- POUs/utils/resetApplication.TcPOU
FUNCTION resetApplication : BOOL
VAR_INPUT    
	pMachine : POINTER TO FB_StateMachine;
END_VAR
VAR
	i 			: INT := 1;
END_VAR

FOR i := 0 TO 6 DO
    GVL.lastErrorsOccurred[i].eventType := E_EventType.None;        // Beispiel für einen "leeren" Event-Typ
    GVL.lastErrorsOccurred[i].severity := E_Severity.Event;         // Standardwert für severity
    GVL.lastErrorsOccurred[i].isTriggered := FALSE;                 // Setzt isTriggered auf FALSE
    GVL.lastErrorsOccurred[i].message := '';                        // Leere Zeichenkette für message
    GVL.lastErrorsOccurred[i].timestamp := DT#1970-01-01-00:00:00;  // Standardzeitstempel (z. B. Unix-Epoche)
    i := i + 1;  
END_FOR;

pMachine^.pd.actor.operatingStateCompressor := FALSE;
pMachine^.pd.actor.operatingStateWaterPump := FALSE;
pMachine^.pd.actor.operatingStateIntermediateCircuitPump := FALSE;
pMachine^.pd.actor.operatingStateLed := FALSE;
pMachine^.pd.actor.openFlowVentil := FALSE;
pMachine^.pd.actor.closeFlowVentil := FALSE;
pMachine^.timerTON(IN := FALSE);

END_FUNCTION

// ---- POUs/FB_StartWaterFlowState.TcPOU
FUNCTION_BLOCK FB_StartWaterFlowState IMPLEMENTS I_State
VAR_INPUT
END_VAR
VAR_OUTPUT
END_VAR
VAR
	pMachine : POINTER TO FB_StateMachine;	
END_VAR

{warning 'Eigenschaftenimplementierung hinzufügen'}
PROPERTY Description : STRING
GET
Description := 'Opening Ventil ...';
END_GET
END_PROPERTY

{warning 'Methodenimplementierung hinzufügen'}
METHOD ErrorDetected : BOOL
VAR_IN_OUT
	errorEvents	: ST_ErrorEvents;
END_VAR
transitionToErrorState(errorEvents := errorEvents, pMachine := pMachine);
END_METHOD

//FB_Init ist immer implizit verfügbar und wird primär für die Initialisierung verwendet.
//Der Rückgabewert wird nicht ausgewertet. Für gezielte Einflussnahme können Sie
//die Methoden explizit deklarieren und darin mit dem Standard-Initialisierungscode 
//zusätzlichen Code bereitstellen. Sie können den Rückgabewert auswerten.
METHOD FB_Init: BOOL
VAR_INPUT    
	bInitRetains: BOOL; // TRUE: Die Retain-Variablen werden initialisiert (Reset warm / Reset kalt)    
	bInCopyCode: BOOL;  // TRUE: Die Instanz wird danach in den Kopiercode kopiert (Online-Change)
	pMachine : POINTER TO FB_StateMachine;
END_VAR
THIS^.pMachine := pMachine;
END_METHOD

{warning 'Methodenimplementierung hinzufügen'}
METHOD HeatIsRequested : BOOL
END_METHOD

METHOD MinWaterFlowReached : BOOL
VAR_INPUT
END_VAR
LogMessage(E_LogType.INFO, 'Ventil ist geöffnet. Durchflussmenge erreicht. Kompressor wird eingeschaltet: -> ', pMachine^.RunningState.Name);
pMachine^.pd.actor.operatingStateWaterPump := TRUE;
pMachine^.pd.actor.operatingStateIntermediateCircuitPump := TRUE;
pMachine^.pd.actor.operatingStateCompressor := TRUE;
pMachine^.SetState(pMachine^.RunningState);
END_METHOD

{warning 'Eigenschaftenimplementierung hinzufügen'}
PROPERTY Name : STRING
GET
Name := 'öffne Ventil';
END_GET
END_PROPERTY

{warning 'Eigenschaftenimplementierung hinzufügen'}
PROPERTY State : E_State
GET
State := E_State.START_WATER_FLOW;
END_GET
END_PROPERTY

{warning 'Methodenimplementierung hinzufügen'}
METHOD TargetTemperatureReached : BOOL
END_METHOD

{warning 'Methodenimplementierung hinzufügen'}
METHOD UserPressedConfirmationButton : BOOL
END_METHOD

METHOD UserPressedSwitchOffButton : BOOL
LogMessage(E_LogType.INFO, 'Aus Button wurde gedrückt -> ', pMachine^.OffState.Name);
switchWaterVentil(bOpen := FALSE, pMachine);
pMachine^.pd.actor.operatingStateCompressor := FALSE;
pMachine^.pd.actor.operatingStateWaterPump := FALSE;
pMachine^.pd.actor.operatingStateIntermediateCircuitPump := FALSE;
pMachine^.SetState(pMachine^.OffState);
END_METHOD

{warning 'Methodenimplementierung hinzufügen'}
METHOD UserPressedSwitchOnButton : BOOL
END_METHOD

{warning 'Methodenimplementierung hinzufügen'}
METHOD WaterHasCooledDown : BOOL
END_METHOD

END_FUNCTION_BLOCK

// ---- POUs/FB_RunningState.TcPOU
FUNCTION_BLOCK FB_RunningState IMPLEMENTS I_State
VAR_INPUT
END_VAR
VAR_OUTPUT
END_VAR
VAR
	pMachine : POINTER TO FB_StateMachine;	
END_VAR

METHOD ActionSwitchOff : BOOL
VAR_INPUT
	message		:	STRING;
END_VAR
pMachine^.timerTON(IN := TRUE, PT := GVL.configValues.minIdleSec);
LogMessage(E_LogType.INFO, message, pMachine^.CoolDownState.Name);
pMachine^.pd.actor.operatingStateCompressor := FALSE;
switchWaterVentil(bOpen := FALSE, pMachine);
pMachine^.pd.sensor.photovoltaicBoost := FALSE;
pMachine^.SetState(pMachine^.CoolDownState);
END_METHOD

PROPERTY Description : STRING
GET
Description := 'Heat pump is running';
END_GET
END_PROPERTY

METHOD ErrorDetected : BOOL
VAR_IN_OUT
	errorEvents		: ST_ErrorEvents;
END_VAR
pMachine^.timerTON(IN := TRUE, PT := GVL.configValues.minIdleSec);
transitionToErrorState(errorEvents := errorEvents, pMachine := pMachine);
END_METHOD

//FB_Init ist immer implizit verfügbar und wird primär für die Initialisierung verwendet.
//Der Rückgabewert wird nicht ausgewertet. Für gezielte Einflussnahme können Sie
//die Methoden explizit deklarieren und darin mit dem Standard-Initialisierungscode 
//zusätzlichen Code bereitstellen. Sie können den Rückgabewert auswerten.
METHOD FB_Init: BOOL
VAR_INPUT    
	bInitRetains: BOOL; // TRUE: Die Retain-Variablen werden initialisiert (Reset warm / Reset kalt)    
	bInCopyCode: BOOL;  // TRUE: Die Instanz wird danach in den Kopiercode kopiert (Online-Change)
	pMachine : POINTER TO FB_StateMachine;
END_VAR
THIS^.pMachine := pMachine;
END_METHOD

METHOD HeatIsRequested : BOOL
END_METHOD

METHOD LimitValuesAreExceeded : BOOL
END_METHOD

METHOD MinWaterFlowReached : BOOL
VAR_INPUT
END_VAR
END_METHOD

PROPERTY Name : STRING
GET
Name := 'Kompressor ein';
END_GET
END_PROPERTY

PROPERTY State : E_State
GET
State := E_State.RUNNING;
END_GET
END_PROPERTY

METHOD TargetTemperatureReached : BOOL
LogMessage(E_LogType.INFO, 'Boiler oben: ', REAL_TO_STRING (pMachine^.pd.sensor.bufferMiddleTemperature));
LogMessage(E_LogType.INFO, 'Zieltemperatur (Ausschalttemperatur): ', REAL_TO_STRING (GVL.configValues.targetTemperatureOff));
LogMessage(E_LogType.INFO, 'Boiler-Ladepumpe: ', BOOL_TO_STRING (pMachine^.pd.sensor.boilerHeatRequest));

ActionSwitchOff('Zieltemperatur erreicht. -> ');
END_METHOD

METHOD UserPressedConfirmationButton : BOOL
END_METHOD

METHOD UserPressedSwitchOffButton : BOOL
ActionSwitchOff('Off Button pressed -> ');
END_METHOD

METHOD UserPressedSwitchOnButton : BOOL
END_METHOD

METHOD WaterHasCooledDown : BOOL
END_METHOD

END_FUNCTION_BLOCK

// ---- POUs/FB_CoolDownState.TcPOU
FUNCTION_BLOCK FB_CoolDownState IMPLEMENTS I_State
VAR_INPUT
END_VAR
VAR_OUTPUT
END_VAR
VAR
	pMachine : POINTER TO FB_StateMachine;	
END_VAR

PROPERTY Description : STRING
GET
Description := 'Heat pump is cooling down';
END_GET
END_PROPERTY

METHOD ErrorDetected : BOOL
VAR_IN_OUT
	errorEvents		: ST_ErrorEvents;
END_VAR
transitionToErrorState(errorEvents := errorEvents, pMachine := pMachine);
END_METHOD

//FB_Init ist immer implizit verfügbar und wird primär für die Initialisierung verwendet.
//Der Rückgabewert wird nicht ausgewertet. Für gezielte Einflussnahme können Sie
//die Methoden explizit deklarieren und darin mit dem Standard-Initialisierungscode 
//zusätzlichen Code bereitstellen. Sie können den Rückgabewert auswerten.
METHOD FB_Init: BOOL
VAR_INPUT    
	bInitRetains: BOOL; // TRUE: Die Retain-Variablen werden initialisiert (Reset warm / Reset kalt)    
	bInCopyCode: BOOL;  // TRUE: Die Instanz wird danach in den Kopiercode kopiert (Online-Change)
	pMachine : POINTER TO FB_StateMachine;
END_VAR
THIS^.pMachine := pMachine;
END_METHOD

METHOD HeatIsRequested : BOOL
END_METHOD

METHOD LimitValuesAreExceeded : BOOL
END_METHOD

METHOD MinWaterFlowReached : BOOL
VAR_INPUT
END_VAR
END_METHOD

PROPERTY Name : STRING
GET
Name := 'abkühlen';
END_GET
END_PROPERTY

PROPERTY State : E_State
GET
State := E_State.COOLDOWN;
END_GET
END_PROPERTY

METHOD TargetTemperatureReached : BOOL
END_METHOD

METHOD UserPressedConfirmationButton : BOOL
END_METHOD

METHOD UserPressedSwitchOffButton : BOOL
LogMessage(E_LogType.INFO, 'Aus Button wurde gedrückt -> ', pMachine^.OffState.Name);
pMachine^.SetState(pMachine^.OffState);
END_METHOD

METHOD UserPressedSwitchOnButton : BOOL
END_METHOD

METHOD WaterHasCooledDown : BOOL
LogMessage(E_LogType.INFO, 'Abkühlungsphase beendet -> ', pMachine^.IdleState.Name);
pMachine^.pd.actor.operatingStateWaterPump := FALSE;
pMachine^.pd.actor.operatingStateIntermediateCircuitPump := FALSE;
pMachine^.SetState(pMachine^.IdleState);
END_METHOD

END_FUNCTION_BLOCK

// ---- POUs/FB_ErrorState.TcPOU
FUNCTION_BLOCK FB_ErrorState IMPLEMENTS I_State
VAR_INPUT
END_VAR
VAR_OUTPUT
END_VAR
VAR
	pMachine : POINTER TO FB_StateMachine;
END_VAR

PROPERTY Description : STRING
GET
Description := 'An error has occurred';
END_GET
END_PROPERTY

METHOD ErrorDetected : BOOL
VAR_IN_OUT
	errorEvents		: ST_ErrorEvents;
END_VAR
// transitionToErrorState(errorEvents := errorEvents, pMachine := pMachine);
END_METHOD

//FB_Init ist immer implizit verfügbar und wird primär für die Initialisierung verwendet.
//Der Rückgabewert wird nicht ausgewertet. Für gezielte Einflussnahme können Sie
//die Methoden explizit deklarieren und darin mit dem Standard-Initialisierungscode 
//zusätzlichen Code bereitstellen. Sie können den Rückgabewert auswerten.
METHOD FB_Init: BOOL
VAR_INPUT    
	bInitRetains: BOOL; // TRUE: Die Retain-Variablen werden initialisiert (Reset warm / Reset kalt)    
	bInCopyCode: BOOL;  // TRUE: Die Instanz wird danach in den Kopiercode kopiert (Online-Change)
	pMachine : POINTER TO FB_StateMachine;
END_VAR
THIS^.pMachine := pMachine;
END_METHOD

METHOD HeatIsRequested : BOOL
END_METHOD

METHOD MinWaterFlowReached : BOOL
VAR_INPUT
END_VAR
END_METHOD

PROPERTY Name : STRING
GET
Name := 'Error';
END_GET
END_PROPERTY

PROPERTY State : E_State
GET
State := E_State.ERROR;
END_GET
END_PROPERTY

METHOD TargetTemperatureReached : BOOL
END_METHOD

METHOD UserPressedConfirmationButton : BOOL
END_METHOD

METHOD UserPressedSwitchOffButton : BOOL
resetApplication(pMachine);
LogMessage(E_LogType.INFO, 'Aus Button wurde gedrückt -> ', pMachine^.OffState.Name);
pMachine^.SetState(pMachine^.OffState);
END_METHOD

METHOD UserPressedSwitchOnButton : BOOL
END_METHOD

METHOD WaterHasCooledDown : BOOL
END_METHOD

END_FUNCTION_BLOCK

// ---- POUs/utils/clearErrorList.TcPOU
FUNCTION clearErrorList : BOOL
VAR
	i 			: INT := 0;
END_VAR


WHILE i <= 6 DO
    GVL.lastErrorsOccurred[i].eventType := E_EventType.None;        // Beispiel für einen "leeren" Event-Typ
    GVL.lastErrorsOccurred[i].severity := E_Severity.Event;         // Standardwert für severity
    GVL.lastErrorsOccurred[i].isTriggered := FALSE;                 // Setzt isTriggered auf FALSE
    GVL.lastErrorsOccurred[i].message := '';                        // Leere Zeichenkette für message
    GVL.lastErrorsOccurred[i].timestamp := DT#1970-01-01-00:00:00;  // Standardzeitstempel (z. B. Unix-Epoche)
    i := i + 1;  
END_WHILE;

END_FUNCTION

// ---- POUs/utils/isVentilOpen.TcPOU
FUNCTION isVentilOpen : BOOL
VAR_INPUT
	pd 		: REFERENCE TO ST_ProcessData;
END_VAR
VAR
END_VAR

isVentilOpen := pd.incident.incidentWaterFlow;

END_FUNCTION

// ---- POUs/utils/toggleIntermediateCircuitPump.TcPOU
FUNCTION toggleIntermediateCircuitPump : BOOL
VAR_INPUT
	pMachine : POINTER TO FB_StateMachine;
END_VAR
VAR
END_VAR

// Das manuelle Ein-Ausschalten der Zwischenkreispumpe ist nur in IDLE oder ERROR Status möglich
IF pMachine^.iState.State = E_State.IDLE OR pMachine^.iState.State = E_State.ERROR THEN
	IF pMachine^.pd.actor.operatingStateIntermediateCircuitPump = FALSE THEN
		LogMessage(E_LogType.INFO, 'Schalte Sole Zwischenkreispumpe: -> ', 'Ein');	
		pMachine^.pd.actor.operatingStateIntermediateCircuitPump := TRUE;
	ELSE
		LogMessage(E_LogType.INFO, 'Schalte Sole Zwischenkreispumpe: -> ', 'Aus');	
		pMachine^.pd.actor.operatingStateIntermediateCircuitPump := FALSE;
	END_IF
END_IF

END_FUNCTION

// ---- POUs/utils/togglePvBoost.TcPOU
FUNCTION togglePvBoost : BOOL
VAR_INPUT
	pMachine : POINTER TO FB_StateMachine;
END_VAR
VAR
END_VAR

IF pMachine^.pd.sensor.photovoltaicBoost = FALSE THEN
	LogMessage(E_LogType.INFO, 'PV Boost wurde geklickt: -> ', 'Ein');	
	pMachine^.pd.sensor.photovoltaicBoost := TRUE;
ELSE
	LogMessage(E_LogType.INFO, 'PV Boost wurde geklickt: -> ', 'Aus');	
	pMachine^.pd.sensor.photovoltaicBoost := FALSE;
END_IF

END_FUNCTION

// ---- POUs/utils/convertTimerToDisplayValue.TcPOU
FUNCTION convertTimerToDisplayValue : INT
VAR_IN_OUT
	timerTon		:	TON;
END_VAR
VAR
END_VAR

convertTimerToDisplayValue := TIME_TO_INT ((GVL.configValues.minIdleSec - timerTon.ET) / 1000);

END_FUNCTION

// ---- POUs/utils/setEventInfo.TcPOU
FUNCTION setEventInfo : BOOL
VAR_INPUT
	events				: REFERENCE TO ST_Events;
	stEvent 			: REFERENCE TO ST_Event;
	isError				: BOOL;
	strMessage 			: STRING(255);
END_VAR

stEvent.message := strMessage;
stEvent.isTriggered := TRUE;
updateEventWithTimestamp(stEvent := stEvent);
events.errorsDetected := isError;

END_FUNCTION

// ---- POUs/utils/updateEventWithTimestamp.TcPOU
FUNCTION updateEventWithTimestamp : DATE_AND_TIME
VAR_INPUT
	stEvent : REFERENCE TO ST_Event;
END_VAR
VAR
	fbSystemTime : GETSYSTEMTIME;
    timeAsFileTime : T_FILETIME;
END_VAR

fbSystemTime(timeLoDW => timeAsFileTime.dwLowDateTime, timeHiDW => timeAsFileTime.dwHighDateTime);
stEvent.timestamp := FILETIME_TO_DT(timeAsFileTime);

END_FUNCTION

// ---- POUs/utils/ScaleAndRoundString.TcPOU
FUNCTION ScaleAndRoundString : String
VAR_INPUT
	realValue 	: REAL;          // Die zu rundende REAL-Zahl
	scaleFactor : INT;           // Rundungsfaktor
END_VAR
VAR
END_VAR

ScaleAndRoundString := REAL_TO_STRING(INT_TO_REAL(REAL_TO_INT(realValue * scaleFactor)) / scaleFactor);

END_FUNCTION

// ---- POUs/utils/calculateTargetTemperatureOn.TcPOU
FUNCTION calculateTargetTemperatureOn : REAL
VAR_INPUT
	photovoltaicSurplus			: BOOL;
	photovoltaicBoost			: BOOL;
END_VAR

IF (photovoltaicSurplus OR photovoltaicBoost) THEN
    calculateTargetTemperatureOn := GVL.configValues.targetTemperatureOnPV;
ELSE
    calculateTargetTemperatureOn := GVL.configValues.targetTemperatureOn;
END_IF;

END_FUNCTION

// ---- POUs/utils/calculateTargetTemperatureOff.TcPOU
FUNCTION calculateTargetTemperatureOff : REAL
VAR_INPUT
	photovoltaicSurplus			: BOOL;
	photovoltaicBoost			: BOOL;
END_VAR

IF (photovoltaicSurplus OR photovoltaicBoost) THEN
    calculateTargetTemperatureOff := GVL.configValues.targetTemperatureOffPV;
ELSE
    calculateTargetTemperatureOff := GVL.configValues.targetTemperatureOff;
END_IF;

END_FUNCTION

// ---- POUs/FB_ProcessData.TcPOU
FUNCTION_BLOCK FB_ProcessData
VAR_INPUT
	pd 				: 	REFERENCE TO ST_ProcessData;
END_VAR
VAR
	sensorRaw		:	ST_SensorRaw; 
END_VAR

(* Temperatur*)
pd.sensor.temperatureEvaporatingIn 		:=	RawToTemperature(sensorRaw.temperatureEvaporatingIn);
pd.sensor.temperatureEvaporatingOut 	:=	RawToTemperature(sensorRaw.temperatureEvaporatingOut);
pd.sensor.temperatureFlow 				:=	RawToTemperature(sensorRaw.temperatureFlow);
pd.sensor.temperatureReturn 			:=	RawToTemperature(sensorRaw.temperatureReturn);
pd.sensor.bufferTopTemperature 			:=	RawToTemperature(sensorRaw.bufferTopTemperature);
pd.sensor.bufferMiddleTemperature 		:=	RawToTemperature(sensorRaw.bufferMiddleTemperature);
pd.sensor.boilerTemperature				:=	RawToTemperature(sensorRaw.boilerTemperature);
pd.sensor.temperatureOverheatedGas 		:=	RawToTemperature(sensorRaw.temperatureOverheatedGas);
pd.sensor.temperatureSourceWaterIn 		:=	RawToTemperature(sensorRaw.temperatureSourceWaterIn);
pd.sensor.temperatureSourceWaterOut 	:=	RawToTemperature(sensorRaw.temperatureSourceWaterOut);

(* Pressure Difference im mBar -  0-10 Volt  or  -10V to +10V *)
pd.sensor.pressureDifferenceEvaporator	:= 	RawToRealAnalog(sensorRaw.pressureDifferenceEvaporator, 0, 200, 10);

(* Pressure in Bar - using 4-20mmA Sensors*)
pd.sensor.pressureHigh	:= 	RawToRealAnalog(sensorRaw.pressureHigh, 0, 18, 10);			(* Range from 0 to 18.0 bar *)
pd.sensor.pressureLow	:= 	RawToRealAnalog(sensorRaw.pressureLow, -0.5, 7, 10);		(* Range from -0.5 to 7.0 bar *)

METHOD RawToRealAnalog : REAL
VAR_INPUT
	rawVal		: INT;
	rawMin		: REAL;
	rawMax		: REAL;	
	roundFactor	: INT;
END_VAR
VAR CONSTANT
	highValue 	: INT := 16#7FFF;  // Hexadezimale Zahl 0x7FFF
END_VAR
VAR
	realVal		: REAL;
END_VAR
realVal := ((rawMax - rawMin) * rawVal) / highValue + rawMin;
RawToRealAnalog := ScaleAndRound(realVal, roundFactor);
END_METHOD

METHOD INTERNAL RawToTemperature : REAL
VAR_INPUT
	raw : INT;
END_VAR
RawToTemperature :=  (INT_TO_REAL (raw)) / 10;
END_METHOD

END_FUNCTION_BLOCK

// ---- POUs/utils/ScaleAndRound.TcPOU
FUNCTION ScaleAndRound : REAL
VAR_INPUT
	realValue 	: REAL;          // Die zu rundende REAL-Zahl
	scaleFactor : INT;           // Rundungsfaktor
END_VAR
VAR
END_VAR

ScaleAndRound := INT_TO_REAL(REAL_TO_INT(realValue * scaleFactor)) / scaleFactor;

END_FUNCTION
